// TwinCAT 3 PLC project pruebaTanque
// ProgramVersion: 3.1.4024.0
// libraries:
//   Tc2_Standard, * (Beckhoff Automation GmbH)
//   Tc2_System, * (Beckhoff Automation GmbH)
//   Tc2_Utilities, * (Beckhoff Automation GmbH)
//   Tc3_Module, * (Beckhoff Automation GmbH)
//   Util, * (System)
//   VisuSymbols,3.5.10.0,System
// project tree:
//   / GlobalTextList.TcGTLO, PlcTask.TcTTO, Visualization Manager.TcVMO (not stored)
//   GVLs/ GVLvars.TcGVL
//   POUs/ MAIN.TcPOU, CalculoTiempoLLenado.TcPOU
//   VISUs/ pantallaHMi.TcVIS
// real-time tasks:
//   TASK PlcTask: cycle T#10ms, priority 20, ADS port 350

CONFIGURATION pruebaTanque
    RESOURCE PLC ON TwinCAT3
        TASK PlcTask(INTERVAL := T#10ms, PRIORITY := 20);
        PROGRAM MAIN WITH PlcTask : MAIN;
    END_RESOURCE
END_CONFIGURATION

// ---- GVLs/GVLvars.TcGVL
{attribute 'qualified_only'}
VAR_GLOBAL
	
	// CUADRO
	{attribute 'OPC.UA.DA' := '1'}
	Start_Button : BOOL;  // Boton de arranque
	{attribute 'OPC.UA.DA' := '1'}
	StopButton : BOOL; // Boton de paro
	{attribute 'OPC.UA.DA' := '1'}
	luzVerde : BOOL; // luz verde stack
	{attribute 'OPC.UA.DA' := '1'}
	luzAmarilla : BOOL; // luz amarilla stack
	{attribute 'OPC.UA.DA' := '1'}
 	luzRoja : BOOL; // luz roja stack
	{attribute 'OPC.UA.DA' := '1'}
	luzBotonStop : BOOL; // luz del boton de stop 
	{attribute 'OPC.UA.DA' := '1'}
	luzBotonStart : BOOL; // luz del boton de start
	{attribute 'OPC.UA.DA' := '1'}
	luzBotonReset : BOOL; // luz boton start
	{attribute 'OPC.UA.DA' := '1'}
	seta : BOOL; // seta de emergencia
	{attribute 'OPC.UA.DA' := '1'}
	resetBoton : BOOL; // Boton de reset (tras rearme de seta)
	
	
	// SENSORES
	{attribute 'OPC.UA.DA' := '1'}   
	Sensor_Tanque_Salida : BOOL;       // Sensor fotoeléctrico justo antes del tanque
//	{attribute 'OPC.UA.DA' := '1'}    
//	Sensor_Barril_Listo  : BOOL;       // Sensor que detecta barril en posición
	//	 {attribute 'OPC.UA.DA' := '1'}    
	

	// TANQUE
	//	Level_Meter          : REAL;       // Nivel del tanque (0-10 V)
	{attribute 'OPC.UA.DA' := '1'}
	// Valvulas tanque
	{attribute 'OPC.UA.DA' := '1'}    
	Fill_Valve           : BOOL;       // Válvula de llenado (0–10 V)
	{attribute 'OPC.UA.DA' := '1'}    
	Discharge_Valve      : BOOL;       // Válvula de salida (0–10 V)
	
	
	
	// CINTAS
	{attribute 'OPC.UA.DA' := '1'}    
	Cinta_Entrada        : BOOL;
	{attribute 'OPC.UA.DA' := '1'}    
	Cinta_Tanque         : BOOL;
	{attribute 'OPC.UA.DA' := '1'}    
	Cinta_Salida         : BOOL;
	

END_VAR

// ---- POUs/MAIN.TcPOU
PROGRAM MAIN
VAR  
	Sensor_Anterior : BOOL := FALSE;
	Flanco_Subida : BOOL := FALSE;
	Estado: INT := 0; // 0: Espera | 1: Descargando | 2: Post-descarga
	
	
	// Variables internas
	Sistema_Activo : BOOL;
	
	Timer_Stop           : TON;
	Esperando_Timer      : BOOL := FALSE;
	
	Nivel_Bajo           : BOOL;
	Nivel_Alto           : BOOL;
	Nivel_OK             : BOOL;
	// Temporizador para la descarga
	Timer_Descarga       : TON;
	Descargando          : BOOL := FALSE;
	Timer_Llenado: TON;
	InicioLLenado: BOOL := TRUE;
	VienesDeDescarga: BOOL;
	primeraVez: BOOL;
	numDescargas: INT;
	luzVerde: BOOL;
	luzAmarilla: BOOL;
	luzRoja: BOOL;
	tiempoLLenado: TIME;
	tiempoTranscurrrido: TIME;
	parado: BOOL; // variable que india que la secucnia paso por el etado de parado (se pulso stop)
	tiempoRestante: DINT;
	emergencia: BOOL;
	luzBotonStart: BOOL;
	luzBotonStop: BOOL;
	luzBotonReset: BOOL;
	tiempoCargaBarril: TIME;
	cargandoTanque: BOOL;
END_VAR

// Luces de los botones del cuadro
// Solo se mantienen encendidas mientras estan pulsados
luzBotonStart := FALSE;
luzBotonStop := FALSE;
luzBotonReset := FALSE;



// Enclavamiento del boton de start
IF GVLvars.Start_Button  AND emergencia = FALSE THEN
    Sistema_Activo := TRUE;
	primeraVez := TRUE;
	luzVerde := TRUE;
	luzAmarilla := FALSE;
	luzRoja := FALSE;
	parado := FALSE;
	emergencia := FALSE;
	luzBotonStart := TRUE;
END_IF

// Boton Stop -> se para 
IF NOT GVLvars.StopButton AND emergencia = FALSE  THEN
	Sistema_Activo := FALSE;
	parado := TRUE;
	luzVerde := FALSE;
	luzAmarilla := TRUE;
	luzRoja := FALSE;
	//tiempoTranscurrrido := Timer_Llenado.ET;
	InicioLLenado := FALSE;
	emergencia := FALSE;
	luzBotonStop := TRUE;
END_IF
 
// Si se acciona la seta de emergencia se para todo
IF GVLvars.seta = false  THEN
	Sistema_Activo := FALSE;
	parado := FALSE;
	luzVerde := FALSE;
	luzAmarilla := FALSE;
	luzRoja := TRUE;
	//tiempoTranscurrrido := Timer_Llenado.ET;
	//InicioLLenado := FALSE;
	emergencia := TRUE;
END_IF

// Si la seta no esta armada pero lo estuvo previamente 
// se debe pulsar el boton de reset para reanudar la actividad 
IF  GVLvars.seta AND emergencia THEN
	IF GVLvars.resetBoton THEN
		Sistema_Activo := TRUE;
		//primeraVez := TRUE;
		luzVerde := TRUE;
		luzAmarilla := FALSE;
		luzRoja := FALSE;
		parado := FALSE;
		emergencia := FALSE;
		luzBotonReset := TRUE;
	END_IF
END_IF


// se pretende que el tanuqe este siempre ente un 20-80%
// si el tanuqe esta vacio se necesitan  39s para el 80% 
// si el tanque esta al 20% se necesitan 31s para el 80%
// si el se paro en algun punto se calcula el tiempo rstante
IF primeraVez THEN
	tiempoLLenado := T#39S;
//ELSIF parado THEN
//	tiempoRestante := TIME_TO_DINT(tiempoLLenado) - TIME_TO_DINT(tiempoTranscurrrido);
//	tiempoLLenado := DINT_TO_TIME(tiempoRestante);
ELSE 
	tiempoLLenado := T#32S;
END_IF

IF Sistema_Activo THEN
	// Control inicial llenado tanque
	Timer_Llenado(IN := InicioLLenado, PT := tiempoLLenado);
	IF NOT Timer_Llenado.Q AND InicioLLenado THEN
		GVLvars.Fill_Valve := TRUE;           // Abrir valvula llenado
		cargandoTanque := TRUE;
	ELSE
		GVLvars.Fill_Valve := FALSE;          // Cerrar valvula llenado
		// Solo dejar de iniciar llenado después de completar timer
		InicioLLenado := FALSE;
		cargandoTanque := FALSE;
	END_IF
END_IF




// FLANCO DE BAJADA del sensor antes del tanque
//Sensor_FlancoBajada := Sensor_Anterior AND NOT GVL_Inputs.Sensor_Tanque_Salida;
//Sensor_Anterior := GVL_Inputs.Sensor_Tanque_Salida;

//// Limites nivel tanque
//Nivel_Bajo := GVL_Inputs.Level_Meter < 2.5;
//Nivel_Alto := GVL_Inputs.Level_Meter > 9.0;
//Nivel_OK   := GVL_Inputs.Level_Meter > 2.5;

//// Control de llenado del tanque
//IF Nivel_Bajo THEN
//    GVL_Inputs.Fill_Valve := 10;  // Abrir completamente valvula entrada
//ELSIF Nivel_Alto THEN
//    GVL_Inputs.Fill_Valve := 0;   // Cerrar valvula
//END_IF

// Si el sistema esta activo
IF Sistema_Activo  AND InicioLLenado=FALSE  AND emergencia = FALSE THEN
	//La oprimera vez que se inica el programa se arrancan las cintas
	IF primeraVez THEN
		GVLvars.Cinta_Entrada := TRUE;
		GVLvars.Cinta_Tanque  := TRUE;
		GVLvars.Cinta_Salida  := TRUE;
		primeraVez := FALSE;
	END_IF


Flanco_Subida := (NOT Sensor_Anterior) AND GVLvars.Sensor_Tanque_Salida;
Sensor_Anterior := GVLvars.Sensor_Tanque_Salida;


    // Máquina de estados
    CASE Estado OF

        // Estado 0: Esperando objeto en la boca del tanque
        0:
			//IF emergencia = FALSE AND cargandoTanque = FALSE THEN
				GVLvars.Cinta_Entrada := TRUE;
				GVLvars.Cinta_Tanque  := TRUE;
				GVLvars.Cinta_Salida  := TRUE;
				GVLvars.Discharge_Valve := FALSE;
				Timer_Descarga(IN := FALSE);
	
				IF Flanco_Subida THEN
					Estado := 1;
				END_IF
			//END_IF
            

        //  Estado 1: Descargando (2 segundos)
        1:
			// si no se encuentra se seta armada o esprando a rearme
            //IF emergencia = FALSE AND cargandoTanque = FALSE THEN
				GVLvars.Cinta_Entrada := FALSE;
				GVLvars.Cinta_Tanque  := FALSE;
				GVLvars.Cinta_Salida  := FALSE;
				GVLvars.Discharge_Valve := TRUE;
				
				tiempoCargaBarril := CalculoTiempoLLenado(Volume_L :=709, Flow_Lps :=0.3543  );
	
				Timer_Descarga(IN := TRUE, PT := T#2s);
	
				IF Timer_Descarga.Q THEN
					Timer_Descarga(IN := FALSE); // Detener timer
					numDescargas := numDescargas + 1;
					Estado := 2;
				END_IF

			//END_IF
			
        // Estado 2: Post-descarga - reactivar cintas
        2:
			//IF emergencia = FALSE THEN
				IF numDescargas < 16 THEN
					GVLvars.Discharge_Valve := FALSE;
					GVLvars.Cinta_Entrada := TRUE;
					GVLvars.Cinta_Tanque  := TRUE;
					GVLvars.Cinta_Salida  := TRUE;
	
					Estado := 0; // Volver a esperar nuevo objeto
				ELSE
					GVLvars.Discharge_Valve := FALSE;
					GVLvars.Cinta_Entrada := FALSE;
					GVLvars.Cinta_Tanque  := FALSE;
					GVLvars.Cinta_Salida  := FALSE;
					InicioLLenado := TRUE;
					numDescargas := 0;
					Estado := 0; // Volver a esperar nuevo objeto
				END_IF
			//END_IF
			
			
		
            
    END_CASE

    // Flanco de bajada inicia la descarga
    //IF Sensor_FlancoBajada AND Nivel_OK THEN
//	//IF GVL_Inputs.Sensor_Tanque_Salida THEN
//	IF Flanco_Subida THEN

//		Descargando := TRUE;
//		//Timer_Descarga(IN := Descargando, PT := T#2s);
//        // Detener cintas inmediatamente
//        GVL_Inputs.Cinta_Entrada := FALSE;
//        GVL_Inputs.Cinta_Tanque  := FALSE;
//        GVL_Inputs.Cinta_Salida  := FALSE;
//    END_IF

	
	
//    // Mientras se esta descargando
//    IF Descargando THEN
//		//Se inicia temporizador
//		Timer_Descarga(IN := Descargando, PT := T#2S);
//        GVL_Inputs.Discharge_Valve := TRUE;  // Abrir valvula del tanque
		
//		// Termina descarga
//        IF Timer_Descarga.Q THEN
//        	// cerrar valvula    
//            GVL_Inputs.Discharge_Valve := FALSE;
//            Descargando := FALSE;
//			VienesDeDescarga := TRUE;

////            // Reactivar cintas
////            GVL_Inputs.Cinta_Entrada := TRUE;
////            GVL_Inputs.Cinta_Tanque  := TRUE;
////            GVL_Inputs.Cinta_Salida  := TRUE;
//        END_IF
//    END_IF

////    // Si no estamos descargando ni se detecta un objeto en la entrada del tanque
//    //IF Descargando = FALSE AND VienesDeDescarga = TRUE THEN
//	IF VienesDeDescarga = TRUE THEN
//        GVL_Inputs.Cinta_Entrada := TRUE;
//        GVL_Inputs.Cinta_Tanque  := TRUE;
//        GVL_Inputs.Cinta_Salida  := TRUE;
//        GVL_Inputs.Discharge_Valve := FALSE	;
//	    VienesDeDescarga := FALSE;
//    END_IF

ELSE
    // Sistema desactivado
    GVLvars.Cinta_Entrada := FALSE;
    GVLvars.Cinta_Tanque  := FALSE;
    GVLvars.Cinta_Salida  := FALSE;
//    GVL_Inputs.Fill_Valve := 0.0;
//    GVL_Inputs.Discharge_Valve := 0.0;
    Timer_Descarga(IN := FALSE);
    Descargando := FALSE;
END_IF



// ------------------------- Actualizar salidas -------------------------

GVLvars.luzAmarilla := luzAmarilla;
GVLvars.luzRoja := luzRoja;
GVLvars.luzVerde := luzVerde;
GVLvars.luzBotonReset := luzBotonReset;
GVLvars.luzBotonStart := luzBotonStart;
GVLvars.luzBotonStop := luzBotonStop;

END_PROGRAM

// ---- POUs/CalculoTiempoLLenado.TcPOU
FUNCTION CalculoTiempoLLenado : TIME
VAR_INPUT
    Volume_L : REAL;
    Flow_Lps : REAL;
END_VAR
VAR
    msTime : UDINT;
	sTime: DINT;
	Flow_m3ps: REAL;
END_VAR

// Tiempo llenado = (volumen barril / caudal tanque)
//IF Flow_Lps > 0 THEN
//    msTime := TRUNC(Volume_L / Flow_Lps * 1000); // milisegundos
//ELSE
//    msTime := 0;
//END_IF

//CalculoTiempoLLenado := T#0MS + msTime * T#1MS; // suma de TIME

// Conversión de caudal: m³/s → L/s
// 1 m³/s = 1000 L/s
Flow_Lps := Flow_m3ps * 1000;

IF Flow_Lps > 0 THEN
    sTime := TRUNC(Volume_L / Flow_Lps); // segundos
ELSE
    sTime := 0;
END_IF

CalculoTiempoLLenado := T#0S + sTime * T#1S; // ahora suma en segundos

END_FUNCTION

// ---- GlobalTextList.TcGTLO
TEXTLIST GlobalTextList
  253 = 'Cargando Elemento'
  638 = 'Cargando Tanque'
  516 = 'Start'
  778 = 'Stop'
END_TEXTLIST

// ---- VISUs/pantallaHMi.TcVIS
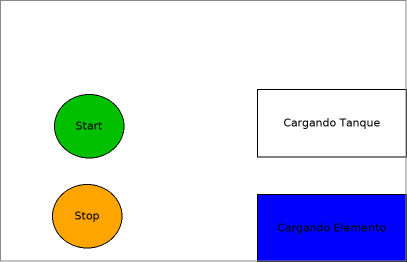
VISUALIZATION pantallaHMi  // 407x262
    Ellipse (54,94 70x64), "Start"
        toggle GVLvars.Start_Button
    Ellipse (52,184 70x64), "Stop"
        toggle GVLvars.StopButton
    RoundedRectangle (257,89 150x68), "Cargando Tanque"
        toggle GVLvars.Fill_Valve
    RoundedRectangle (257,194 150x68), "Cargando Elemento"
        toggle GVLvars.Discharge_Valve
END_VISUALIZATION
